% RSLogix 500 project AT_LAB2 (DEBOUNCE).RSS, saved by version 12.00.00.00 %
PROJECT "UNTITLED"    % processor: Bul.1763 MicroLogix 1100 Series A %

PROGRAM FILES
  LAD 2   5 rungs

DATA FILES
  O0 OUTPUT  4 elements
  I1 INPUT  6 elements
  S2 STATUS  66 elements
  B3 BINARY  1 elements
  T4 TIMER  1 elements
  C5 COUNTER  1 elements
  R6 CONTROL  1 elements
  N7 INTEGER  1 elements
  F8 FLOAT  1 elements

LADDER 2
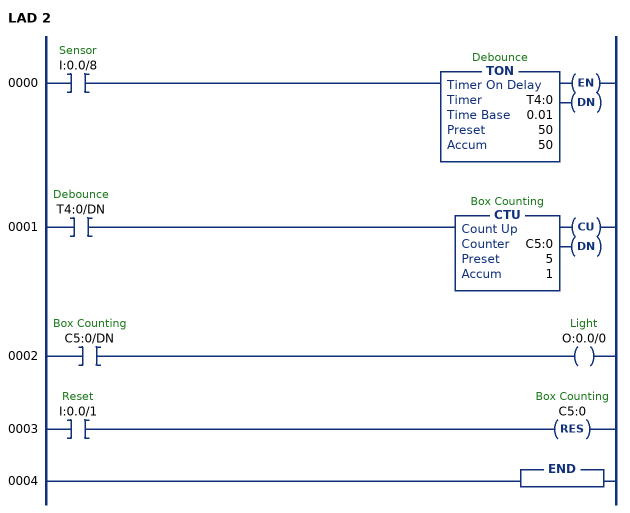
% Rung: 0 %
SOR XIC I:0.0/8 TON T4:0 0.01 50 50 EOR
%   I:0.0/8  "Sensor" %
%   T4:0  "Debounce" %
% Rung: 1 %
SOR XIC T4:0/DN CTU C5:0 5 1 EOR
%   T4:0  "Debounce" %
%   C5:0  "Box Counting" %
% Rung: 2 %
SOR XIC C5:0/DN OTE O:0.0/0 EOR
%   C5:0  "Box Counting" %
%   O:0.0/0  "Light" %
% Rung: 3 %
SOR XIC I:0.0/1 RES C5:0 EOR
%   I:0.0/1  "Reset" %
%   C5:0  "Box Counting" %
% Rung: 4 %
SOR END EOR

DATA TABLE (non-zero values as saved)
DATA T4
% .PRE .ACC %
% T4:0 % 50 50
DATA C5
% .PRE .ACC %
% C5:0 % 5 1
